TYPE ST_ParamStatus :
STRUCT
	eMMA : E_ModeMMA; 
	xModePasAPas:BOOL;
	xErreur:BOOL;
	xInitOk:BOOL;//indique que l'initialisation a été exécutée
END_STRUCT
END_TYPE

(* stored: Version 1.1.0.1, ProductVersion 3.1.4020.6
   DUT ST_ParamStatus: Id {e06697d4-ad48-4213-8945-0ad60333984b} *)
